RoboDK station: New Station (1).rdk

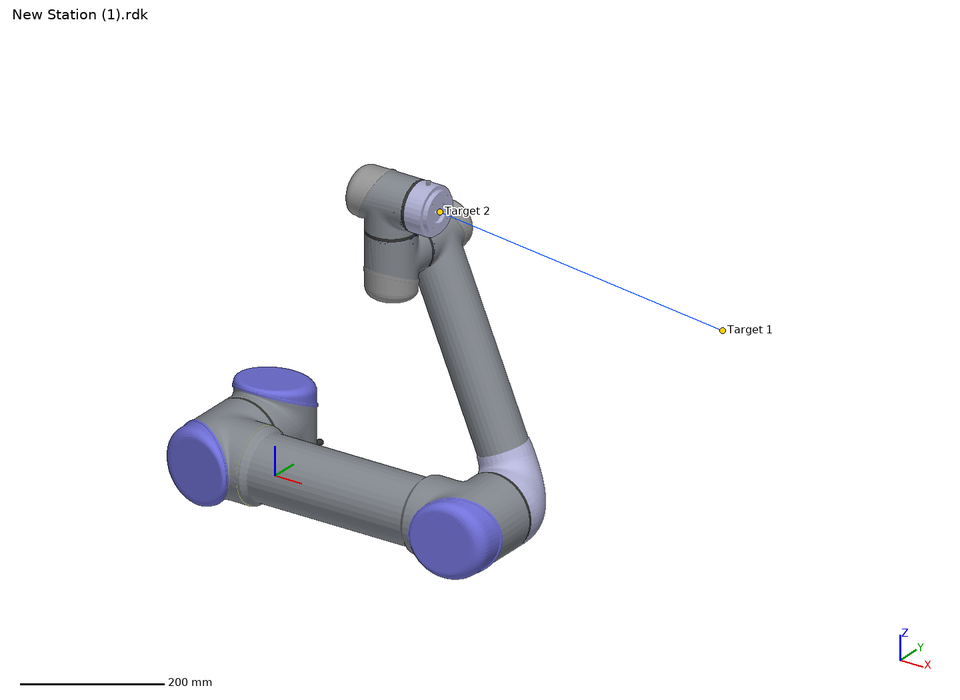
[picture v0: the station drawn from its stored meshes, robots at their saved joint values, targets as dots, program paths as lines]
Station New Station (1). Poses are relative to the parent item; angles as X-Y-Z fixed-axis rotations.
  - frame UR5 Base at (0, 0, 0) mm
    - robot UR5: 6 axes, payload 5 kg, reach 850 mm, repeatability 0.1 mm, weight 18.4 kg
        modified DH rows (alpha deg, a mm, theta deg, d mm): 0, 0, 0, 89.2; 90, 0, 180, 0; 0, 425, 0, 0; 0, 392.43, 0, 109; -90, 0, 0, 93.65; 90, 0, 180, 82
        joint limits [-360, -360, -360, -360, -360, -360] to [360, 360, 360, 360, 360, 360]; home [0, -90, -90, 0, 90, 0]; saved at [0, 180.558, -247.77, -112.789, 90, 0]
    - target Target 1 (Cartesian target) at (832.69, -109, 499.71) mm, rotated rx -90 ry 0 rz -90 deg; joints [0, -152.721, -9.154, -18.124, 90, 0] of UR5
    - target Target 2 (Cartesian target) at (354.98, -109, 548.79) mm, rotated rx -90 ry 0 rz -90 deg; joints [0, 180.558, -247.77, -112.789, 90, 0] of UR5
  - program Prog1 (3 instructions, listed below)
  - Python program Prog2 (listed below)

--- program Prog1 (robot UR5) ---
  Set Ref.: UR5 Base
  MoveJ (Target 1)
  MoveJ (Target 2)

--- Python program Prog2 ---
# This macro shows an example to draw a polygon of radius R and n_sides vertices using the RoboDK API for Python
from robolink import *    # API to communicate with RoboDK for simulation and offline/online programming
from robodk import *      # Robotics toolbox for industrial robots

# Any interaction with RoboDK must be done through RDK:
RDK = Robolink()

# Select a robot (popup is displayed if more than one robot is available)
robot = RDK.ItemUserPick('Select a robot', ITEM_TYPE_ROBOT)
if not robot.Valid():
    raise Exception('No robot selected or available')


# get the current position of the TCP with respect to the reference frame:
# (4x4 matrix representing position and orientation)
target_ref = robot.Pose()
pos_ref = target_ref.Pos()
print("Drawing a polygon around the target: ")
print(Pose_2_TxyzRxyz(target_ref))


# move the robot to the first point:
robot.MoveJ(target_ref)

# It is important to provide the reference frame and the tool frames when generating programs offline
robot.setPoseFrame(robot.PoseFrame())
robot.setPoseTool(robot.PoseTool())
robot.setZoneData(10) # Set the rounding parameter (Also known as: CNT, APO/C_DIS, ZoneData, Blending radius, cornering, ...)
robot.setSpeed(200) # Set linear speed in mm/s

# Set the number of sides of the polygon:
n_sides = 6
R = 100

# make a hexagon around reference target:
for i in range(n_sides+1):
    ang = i*2*pi/n_sides #angle: 0, 60, 120, ...

    #-----------------------------
    # Movement relative to the reference frame
    # Create a copy of the target
    target_i = Mat(target_ref)
    pos_i = target_i.Pos()
    pos_i[0] = pos_i[0] + R*cos(ang)
    pos_i[1] = pos_i[1] + R*sin(ang)
    target_i.setPos(pos_i)
    print("Moving to target %i: angle %.1f" % (i, ang*180/pi))
    print(str(Pose_2_TxyzRxyz(target_i)))
    robot.MoveL(target_i)

    #-----------------------------
    # Post multiply: relative to the tool
    #target_i = target_ref * rotz(ang) * transl(R,0,0) * rotz(-ang)
    #robot.MoveL(target_i)

# move back to the center, then home:
robot.MoveL(target_ref)

print('Done')
